// TIA Portal V16 export
// export: Created 2020-03-29T17:41:51.5680055Z, ExportSetting None, DisplayName Totally Integrated Automation Portal, DisplayVersion V16 Update 1, DisplayName TIA Portal Version Control Interface, DisplayVersion V16, DisplayName TIA Portal Openness, DisplayVersion V16 Update 1, DisplayName SINAMICS Startdrive Advanced, DisplayVersion V16 Update 1, DisplayName SINAMICS Startdrive G130, G150, S120, S150, SINAMICS MV, S210, DisplayVersion V16 Update 1, DisplayName SINAMICS Startdrive G110M, G120, G120C, G120D, G120P, DisplayVersion V16 Update 1, DisplayName STEP 7 Professional, DisplayVersion V16 Update 1, DisplayName STEP 7 Safety, DisplayVersion V16, DisplayName WinCC Advanced, DisplayVersion V16 Update 1
FUNCTION_BLOCK "Valve"   // FB1, LAD
TITLE = Valve control
{ S7_Optimized_Access := 'TRUE' }
// easy sample
// stored: MemoryReserve 100, SetENOAutomatically false
   VAR_INPUT
      Release : Bool;
      OpenValve : Bool;
      CloseValve : Bool;
   END_VAR
   VAR_OUTPUT
      Valve : Bool;
   END_VAR
   VAR
      StateValve : Bool;
   END_VAR
BEGIN

REGION Network 1: Open valve
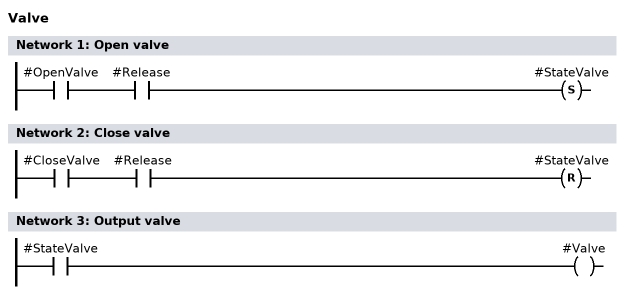
   RUNG wire#powerrail
      Contact( #OpenValve )
      Contact( #Release )
      S_Coil( #StateValve )
   END_RUNG
   // the same network as SCL:
   IF #OpenValve AND #Release THEN #StateValve := TRUE; END_IF;
END_REGION

REGION Network 2: Close valve
   RUNG wire#powerrail
      Contact( #CloseValve )
      Contact( #Release )
      R_Coil( #StateValve )
   END_RUNG
   // the same network as SCL:
   IF #CloseValve AND #Release THEN #StateValve := FALSE; END_IF;
END_REGION

REGION Network 3: Output valve
   RUNG wire#powerrail
      Contact( #StateValve )
      Coil( #Valve )
   END_RUNG
   // the same network as SCL:
   #Valve := #StateValve;
END_REGION
END_FUNCTION_BLOCK
